// Function block with methods demonstrating TwinCAT 3 OOP features

FUNCTION_BLOCK FB_WithMethods

VAR_INPUT
    bEnable : BOOL;
END_VAR

VAR_OUTPUT
    bDone : BOOL;
    nStatus : INT;
END_VAR

VAR
    nInternalState : INT := 0;
    fValue : REAL := 0.0;
END_VAR

// Main execution logic
IF bEnable THEN
    nInternalState := nInternalState + 1;
END_IF;

// Method: Initialize
// Initializes the function block state

METHOD Initialize : BOOL

VAR_INPUT
    bReset : BOOL := FALSE;
    nInitValue : INT := 0;
END_VAR

VAR
    bLocalFlag : BOOL;
END_VAR
// Initialize method implementation
IF bReset THEN
    nInternalState := nInitValue;
    fValue := 0.0;
    bLocalFlag := TRUE;
END_IF;

Initialize := bLocalFlag;
END_METHOD

// Method: GetStatus
// Returns the current status

METHOD PUBLIC GetStatus : INT

VAR_INPUT
    bDetailed : BOOL := FALSE;
END_VAR

VAR
    nTempStatus : INT;
END_VAR
// GetStatus method implementation
nTempStatus := nInternalState;

IF bDetailed AND nInternalState > 0 THEN
    nTempStatus := nTempStatus * 10;
END_IF;

GetStatus := nTempStatus;
END_METHOD

// Method: ProcessData
// Processes data with loops

METHOD PRIVATE ProcessData : REAL

VAR_INPUT
    anData : ARRAY[0..9] OF INT;
END_VAR

VAR
    i : INT;
    fSum : REAL := 0.0;
END_VAR
// ProcessData method with FOR loop
FOR i := 0 TO 9 DO
    fSum := fSum + INT_TO_REAL(anData[i]);
END_FOR;

ProcessData := fSum;
END_METHOD

END_FUNCTION_BLOCK

(* stored: Version 1.1.0.1
   POU FB_WithMethods: Id {aaaaaaaa-bbbb-cccc-dddd-eeeeeeeeeeee}, SpecialFunc None
   Method Initialize: Id {11111111-2222-3333-4444-555555555555}
   Method GetStatus: Id {22222222-3333-4444-5555-666666666666}
   Method ProcessData: Id {33333333-4444-5555-6666-777777777777} *)
